Omron CX-Programmer project NewProject (CX-Programmer 9.61)

# PLC PLC1: CP1H XA

## Global symbols (name address type ; comment)
0.00 BOOL  ; Start
0.01 BOOL  ; Stop
0.02 BOOL  ; D1
0.03 BOOL  ; D2
0.04 BOOL  ; BoxEmitSwitch
0.05 BOOL  ; Det
0.06 BOOL  ; D3
100.00 BOOL  ; M0
100.01 BOOL  ; M1
10.00 BOOL  ; 6m
10.01 BOOL  ; 2m1
10.02 BOOL  ; 2m2
10.03 BOOL  ; MZ
10.04 BOOL  ; Emitter
10.05 BOOL  ; Stoper
10.06 BOOL  ; Grab
10.07 BOOL  ; MX
T0000 BOOL  ; Tim1

## Program NewProgram1 (cyclic task 0)

### Section Section1

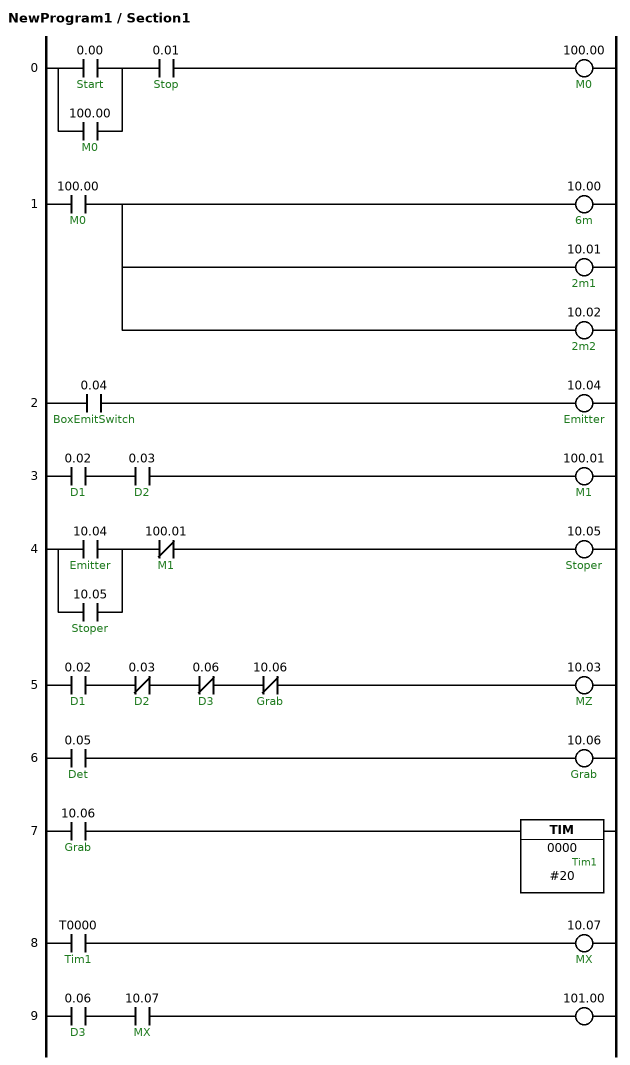
; rung 0
LD 0.00  ; Start
OR 100.00  ; M0
AND 0.01  ; Stop
OUT 100.00  ; M0
; rung 1
LD 100.00  ; M0
OUT 10.00  ; 6m
OUT 10.01  ; 2m1
OUT 10.02  ; 2m2
; rung 2
LD 0.04  ; BoxEmitSwitch
OUT 10.04  ; Emitter
; rung 3
LD 0.02  ; D1
AND 0.03  ; D2
OUT 100.01  ; M1
; rung 4
LD 10.04  ; Emitter
OR 10.05  ; Stoper
ANDNOT 100.01  ; M1
OUT 10.05  ; Stoper
; rung 5
LD 0.02  ; D1
ANDNOT 0.03  ; D2
ANDNOT 0.06  ; D3
ANDNOT 10.06  ; Grab
OUT 10.03  ; MZ
; rung 6
LD 0.05  ; Det
OUT 10.06  ; Grab
; rung 7
LD 10.06  ; Grab
TIM 0000 #20  ; Tim1
; rung 8
LD T0000  ; Tim1
OUT 10.07  ; MX
; rung 9
LD 0.06  ; D3
AND 10.07  ; MX
OUT 101.00

### Section END
; rung 0
END(001)